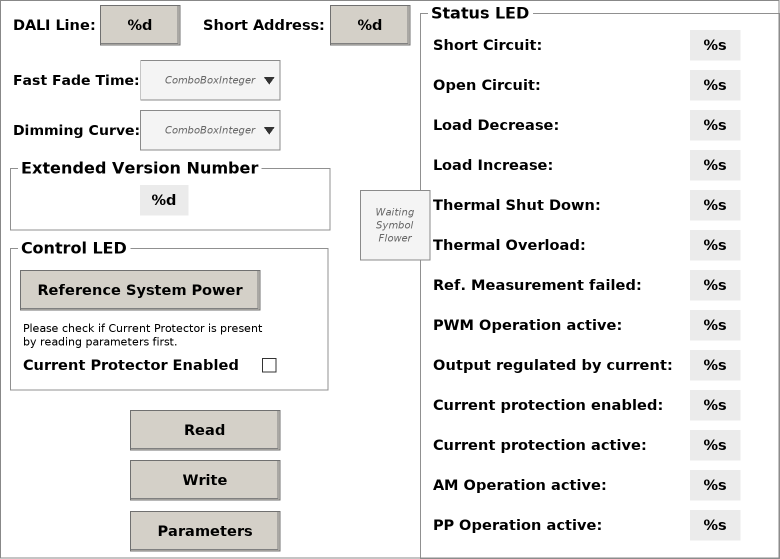
VISUALIZATION Visu_Part207Status  // 780x559
    GroupBox (420,5 360x554), "Status LED"
        Textfield (10,25 250x30), "Short Circuit:"
        Textfield (10,65 250x30), "Open Circuit:"
        Textfield (10,105 250x30), "Load Decrease:"
        Textfield (270,25 50x30), "%s", text variable: DALI_Commissioning.fbPart207StatusLED.sShortCircuit
        Textfield (270,65 50x30), "%s", text variable: DALI_Commissioning.fbPart207StatusLED.sOpenCircuit
        Textfield (270,105 50x30), "%s", text variable: DALI_Commissioning.fbPart207StatusLED.sLoadDecrease
        Textfield (10,145 250x30), "Load Increase:"
        Textfield (270,145 50x30), "%s", text variable: DALI_Commissioning.fbPart207StatusLED.sLoadIncrease
        Textfield (10,345 250x30), "Output regulated by current:", invisible if: DALI_Commissioning.fbPart207StatusLED.bInvisible
        Textfield (10,385 250x30), "Current protection enabled:", invisible if: DALI_Commissioning.fbPart207StatusLED.bInvisible
        Textfield (10,425 250x30), "Current protection active:", invisible if: DALI_Commissioning.fbPart207StatusLED.bInvisible
        Textfield (10,185 250x30), "Thermal Shut Down:"
        Textfield (10,225 250x30), "Thermal Overload:"
        Textfield (10,265 250x30), "Ref. Measurement failed:"
        Textfield (10,465 250x30), "AM Operation active:", invisible if: DALI_Commissioning.fbPart207StatusLED.bInvisible
        Textfield (10,505 250x30), "PP Operation active:", invisible if: DALI_Commissioning.fbPart207StatusLED.bInvisible
        Textfield (10,305 250x30), "PWM Operation active:", invisible if: DALI_Commissioning.fbPart207StatusLED.bInvisible
        Textfield (270,225 50x30), "%s", text variable: DALI_Commissioning.fbPart207StatusLED.sThermalOverload
        Textfield (270,425 50x30), "%s", text variable: DALI_Commissioning.fbPart207StatusLED.sCurrentProtectorActive, invisible if: DALI_Commissioning.fbPart207StatusLED.bInvisible
        Textfield (270,385 50x30), "%s", text variable: DALI_Commissioning.fbPart207StatusLED.sCurrentProtectorEnabled, invisible if: DALI_Commissioning.fbPart207StatusLED.bInvisible
        Textfield (270,345 50x30), "%s", text variable: DALI_Commissioning.fbPart207StatusLED.sOutputCurrentControlled, invisible if: DALI_Commissioning.fbPart207StatusLED.bInvisible
        Textfield (270,465 50x30), "%s", text variable: DALI_Commissioning.fbPart207StatusLED.sAMOperation, invisible if: DALI_Commissioning.fbPart207StatusLED.bInvisible
        Textfield (270,505 50x30), "%s", text variable: DALI_Commissioning.fbPart207StatusLED.sPowerPulseOperation, invisible if: DALI_Commissioning.fbPart207StatusLED.bInvisible
        Textfield (270,265 50x30), "%s", text variable: DALI_Commissioning.fbPart207StatusLED.sReferenceMeasurementFailed
        Textfield (270,185 50x30), "%s", text variable: DALI_Commissioning.fbPart207StatusLED.sThermalShutDown
        Textfield (270,305 50x30), "%s", text variable: DALI_Commissioning.fbPart207StatusLED.sPWMOperation, invisible if: DALI_Commissioning.fbPart207StatusLED.bInvisible
    Button (130,460 150x40), "Write"
        OnMouseClick: execute { DALI_Commissioning.fbPart207StatusLED.bWrite := TRUE; }
    GroupBox (10,240 318x150), "Control LED"
        Textfield (10,110 230x30), "Current Protector Enabled", invisible if: NOT DALI_Commissioning.fbPart207ParametersLED.bQueryCurrentProtectionDevicePresent
        Checkbox (250,110 30x30), variable: DALI_Commissioning.fbPart207StatusLED.bCurrentProtector, invisible if: NOT DALI_Commissioning.fbPart207ParametersLED.bQueryCurrentProtectionDevicePresent, input disabled if: DALI_Commissioning.fbPart207ParametersLED.bQueryCurrentProtectionDevicePresent
        Button (10,30 240x40), "Reference System Power"
            OnMouseClick: execute { DALI_Commissioning.fbPart207StatusLED.bReferenceSystempower := TRUE; }
        Label (10,80 300x30), "Please check if Current Protector is present by reading parameters first."
    Button (130,410 150x40), "Read"
        OnMouseClick: execute { DALI_Commissioning.fbPart207StatusLED.bRead := TRUE; }
    WaitingSymbolFlower (360,190 70x70), invisible if: DALI_Commissioning.fbPart207StatusLED.bHideWaitSymbol
    GroupBox (10,160 320x70), "Extended Version Number"
        Textfield (130,25 48x30), "%d", text variable: DALI_Commissioning.fbPart207StatusLED.nExtendedVersionNumber
    Button (130,511 150x40), "Parameters"
        OnMouseClick: change screen: Visu_Part207Parameters
    Group (200,5 210x40)
        Textfield (0,0 130x40), "Short Address:"
        Button (130,0 80x40), "%d", text variable: DALI_Commissioning.fbPart207StatusLED.nAddress
            OnMouseClick: write the text variable via Default, min 0, max 63, title "Insert Short Address"
    Group (10,110 270x40)
        Textfield (0,0 130x40), "Dimming Curve:"
        ComboBoxInteger (130,0 140x40), variable: DALI_Commissioning.fbPart207StatusLED.eDimmingCurve, text list: 'DimmingCurve'
    Group (10,60 270x40)
        ComboBoxInteger (130,0 140x40), variable: DALI_Commissioning.fbPart207StatusLED.eFastFadeTime, text list: 'FastFadeTime'
        Textfield (0,0 130x40), "Fast Fade Time:"
    Group (10,5 170x40)
        Textfield (0,0 110x40), "DALI Line:"
        Button (90,0 80x40), "%d", text variable: GVL_Internal.nDALILine
            OnMouseClick: write the text variable via Default, min 1, max 10, title "Choose line"
END_VISUALIZATION

(* stored: Version 1.1.0.1, ProductVersion 3.1.4024.9
   Visu Visu_Part207Status: Id {3fdb9a69-24e2-43b5-83d3-017cfcbce496} *)
